{attribute 'qualified_only'}
VAR_GLOBAL
END_VAR

(* stored: Version 1.1.0.1, ProductVersion 3.1.4022.7
   GVL GVL_02_Parameter_Step_Motor_BOX_Y: Id {65a6c55c-c947-43d1-a4f3-e00a87df385d} *)
